PROGRAM P_UML_Grafcet_Sequence
VAR
END_VAR

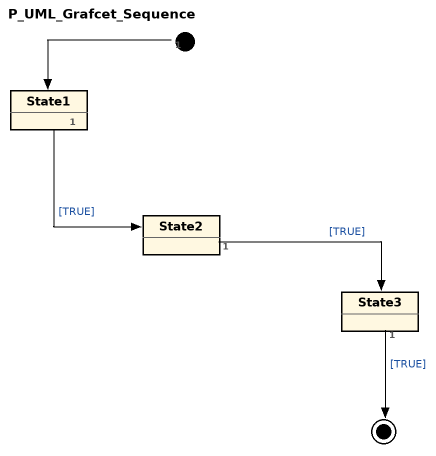
STATECHART P_UML_Grafcet_Sequence  // abortable
    START StartState1
    STATE State1
    STATE State2
    STATE State3
    END EndState1
    StartState1 -> State1  // priority 1, on completion
    State1 -> State2 [TRUE] // priority 1
    State2 -> State3 [TRUE] // priority 1
    State3 -> EndState1 [TRUE] // priority 1
END_STATECHART

END_PROGRAM

(* stored: Version 1.1.0.1, ProductVersion 3.1.4024.5
   POU P_UML_Grafcet_Sequence: Id {aacf82b7-4987-4e0a-aa0e-461f702a75a5}, SpecialFunc None *)
